FUNCTION FUN_ComputeMovingSetPoint : REAL
VAR_INPUT
	currentTemp 		: REAL;
	targetSetPoint 		: REAL;
END_VAR	
VAR
	deltaTemp 			: REAL;
	sign				: REAL;
	maxDeltaTemp		: REAL;
END_VAR

deltaTemp := targetSetPoint - currentTemp;
maxDeltaTemp := 10.0;

IF deltaTemp >= 0 THEN
	sign := 1.0;
ELSE
	sign := -1.0;
END_IF

IF ABS(deltaTemp) > maxDeltaTemp THEN
	FUN_ComputeMovingSetPoint := sign*maxDeltaTemp + currentTemp;
ELSE
	FUN_ComputeMovingSetPoint := targetSetPoint;
END_IF

END_FUNCTION

(* stored: Version 1.1.0.1, ProductVersion 3.1.4022.7
   POU FUN_ComputeMovingSetPoint: Id {2bde4663-6738-4648-b570-8ccbfe30ee14}, SpecialFunc None *)
